FUNCTION_BLOCK SFC2 (* Basic Function Block Type *)
  (* Standard: 61499-2 *)
  (* Version 0.2, 2003-12-04, JHC, Rockwell Automation, Renamed for better indexing. *)
  (* Version 0.1, 2002-11-05, JHC, Rockwell Automation, Corrected missing ST element in Algorithm REQ. *)
  (* Version 0.0, 2000-05-30, JHC, Rockwell Automation *)
  (* Compiler header: package fb.rt.pnp; *)
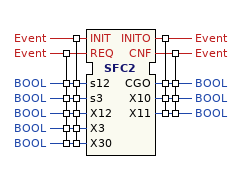
  EVENT_INPUT
    INIT WITH s12, s3, X12, X3, X30; (* Initialization Request *)
    REQ WITH s12, X12, X3, X30, s3; (* Normal Execution Request *)
  END_EVENT
  EVENT_OUTPUT
    INITO WITH CGO, X10, X11; (* Initialization Confirm *)
    CNF WITH CGO, X11, X10; (* Execution Confirmation *)
  END_EVENT
  VAR_INPUT
    s12 : BOOL; (* Input event qualifier *)
    s3 : BOOL;
    X12 : BOOL;
    X3 : BOOL;
    X30 : BOOL;
  END_VAR
  VAR_OUTPUT
    CGO : BOOL; (* Output event qualifier *)
    X10 : BOOL;
    X11 : BOOL;
  END_VAR
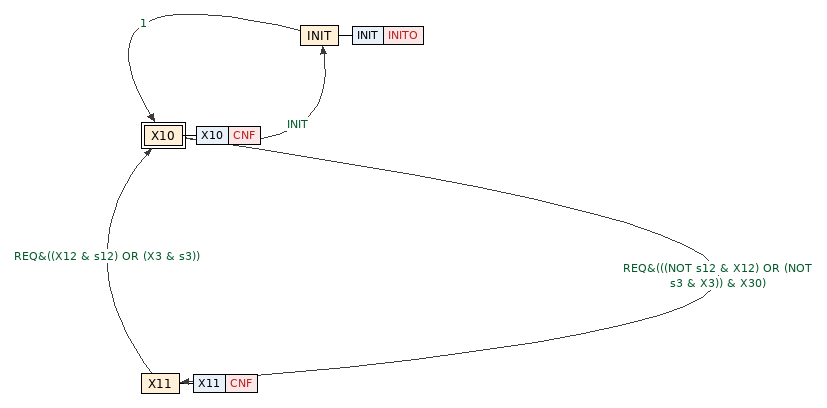
  EC_STATES
    X10 : X10 -> CNF; (* Initial State *)
    INIT : INIT -> INITO; (* Initialization *)
    X11 : X11 -> CNF; (* Normal execution *)
  END_STATES
  EC_TRANSITIONS
    X10 TO INIT := INIT;
    INIT TO X10 := 1;
    X10 TO X11 := REQ&(((NOT s12 & X12) OR (NOT s3 & X3)) & X30);
    X11 TO X10 := REQ&((X12 & s12) OR (X3 & s3));
  END_TRANSITIONS
  ALGORITHM INIT IN ST: (* Initialization algorithm *)
CGO:=false;
X10:=false;
X11:=false;
System.out.println("SFC2: INIT");
  END_ALGORITHM
  ALGORITHM REQ IN ST: (* Normally executed algorithm *)

  END_ALGORITHM
  ALGORITHM X11 IN ST:
CGO:= true;
X10:=false;
X11:=true;
System.out.println("SFC2: X11");
  END_ALGORITHM
  ALGORITHM IntStep IN ST:
CGO:= false;
X11:=false;
System.out.println("SFC2: IntStep");
  END_ALGORITHM
  ALGORITHM X10 IN ST:
X10:=true;
CGO:= false;
X11:=false;
System.out.println("SFC2: X10");
  END_ALGORITHM
END_FUNCTION_BLOCK
